// TIA Portal V19 export
DATA_BLOCK "DB_NSP"   // DB96
{ S7_Optimized_Access := 'FALSE' }
// stored: AutoNumber false
   VAR RETAIN
      Anz_Per_Cyc : Int := 10;   // * Anzahl Positionen pro Zyklus (kleiner eine Sekunde müssen alle durch sein)
      Offset : Int := 20;   // Beginn Datenblock
      leng : Int := 20;   // Länge einer Struktue
      akt_NSP : Int := 55;   // aktueller Eintrag
      Test_on : Bool := TRUE;   // Testfunktion aktiv (nicht gewählte NSP/SPR aus)
      Test_akt : Bool := FALSE;   // Test Einzelpos (TestNr) aktiv
      Test_start : Bool := FALSE;   // Test angemeldet erster Umlauf alles aus
      Sekunde : Bool := FALSE;   // Sekunde M2.5 war ein
      Takt : Bool := FALSE;   // Takt (Sekunde) Zeiten zählen
      AMS_Reset : Bool := FALSE;   // Reset gefordert
      AMS_new : Bool := FALSE;   // Meldung neu schicken
      SammelWarn : Bool := FALSE;   // SammelWarnung min/max über alle Pos.
      Sammelstoer : Bool := FALSE;   // Sammelstörung Timeout über alle Pos.
      noMD_opt_max : Bool := FALSE;   // Überlauf nicht optisch melden
      noMD_opt_min : Bool := FALSE;   // Niveau min nicht optisch melden
      noMD_opt_Zeit : Bool := FALSE;   // Zeitüberschreit. nicht optisch melden
      noMD_aku_max : Bool := FALSE;   // Überlauf nicht akustisch melden
      noMD_aku_min : Bool := FALSE;   // Niveau min nicht akustisch melden
      noMD_aku_Zeit : Bool := FALSE;   // Zeitüberschreit. nicht akustisch melden
      Reset : Bool := FALSE;   // Reset Timeout NS
      TestNr : Int := 0;   // Nachspeisung für Test (alle anderen werden nicht bearbeitet)
      temp_Warn : Bool := FALSE;
      temp_STM : Bool := FALSE;
      resX122 : Bool := FALSE;
      resX123 : Bool := FALSE;
      resX124 : Bool := FALSE;
      resX125 : Bool := FALSE;
      resX126 : Bool := FALSE;
      resX127 : Bool := FALSE;
      resB1 : Byte := 16#00;
      resW1 : Int := 0;
      resD1 : DInt := 0;
      NSP : Array[1..30] of Struct
         NSP : Bool;   // Niveauregelung
         NST_in : Bool;   // Takt nach WT im Bad eingesetzt
         NST_out : Bool;   // Takt nach WT aus Bad ausgehoben
         SPR_in : Bool;   // Spritzen bei FW senkt
         SPR_out : Bool;   // Spritzen bei FW hebt
         SPR_expo : Bool;   // Spritzen während Expozeit
         SPR_Zeit : Bool;   // Spritzen feste Zeit nach Ausheben oder Einsetzen
         resTyp1 : Bool;   // ReserveTyp
         resTyp2 : Bool;   // ReserveTyp
         resTyp3 : Bool;   // ReserveTyp
         resTyp4 : Bool;   // ReserveTyp
         resTyp5 : Bool;   // ReserveTyp
         resTyp6 : Bool;   // ReserveTyp
         resTyp7 : Bool;   // ReserveTyp
         resTyp8 : Bool;   // ReserveTyp
         resTyp9 : Bool;   // ReserveTyp
         Freigabe : Bool;   // Freigabe Nachspeisung
         extern_Start : Bool;   // externe Aktivierung Taktung (zum Beispiel bei mehreren Pos)
         Niveau_ok : Bool;   // Niveau is ok Nachspeisung über Niveauregelung aus
         Nachspeisen : Bool;   // Nachspeisung aktiv --> Ventil auf / Pumpe an
         Spritzen : Bool;   // Spritzregister ein
         AL_Ueberlauf : Bool;   // Behälter Überlauf
         AL_Niv_min : Bool;   // Niveau zu niedrig --> Behälter leer
         AL_Zeit : Bool;   // Nachspeise-Zeitüberschreitung
         Restzeit_NSP : Int;   // Restzeit Nachspeisung
         TestNSP : Int;   // Testzeit Nachspeisung
         Restzeit_SPR : Int;   // Restzeit Spritzen
         VerzT : Int;   // Verzögerung Alarm Überlauf/Min-Niveau
         RestVerz : Int;   // Restzeit bis Alarm
         VerzNS_AL : Int;   // Verzögerung Alarm Nachspeisezeit zu gross
         RestNS_AL : Int;   // Restzeit bis Alarm
         AM_AL_min : Bool;   // Altmerker Alarm min
         AM_AL_Uel : Bool;   // Altmerker Alarm voll
         AM_AL_Zeit : Bool;   // Altmerker Alarm Nachspeise-Zeitüberschreitung
         AM_Bad_belegt : Bool;   // Altmerker Bad belegt
         AM_Reset : Bool;   // Altmerker RESET Nachspeise-Zeitüberschreitung
         res2 : Bool;
         res3 : Bool;
         res4 : Bool;
         SprFree : Bool;   // Spritzregister nicht bedienen (keine Ausgabe weder on noch off) Bedienung ext.
         NSPFree : Bool;   // Nachspeisung nicht bedienen (keine Ausgabe weder on noch off) Bedienung extern
         Warte_NSPT : Bool;   // getaktete Nachspeisung nicht abarbeiten
         res8 : Bool;
         res9 : Bool;
         res10 : Bool;
         res11 : Bool;
         res12 : Bool;
      END_STRUCT;
   END_VAR
BEGIN
   NSP[1..30].NSP := FALSE;
   NSP[1..30].NST_in := FALSE;
   NSP[1..30].NST_out := FALSE;
   NSP[1..30].SPR_in := FALSE;
   NSP[1..25].SPR_out := FALSE;
   NSP[26].SPR_out := TRUE;
   NSP[27..29].SPR_out := FALSE;
   NSP[30].SPR_out := TRUE;
   NSP[1..30].SPR_expo := FALSE;
   NSP[1..30].SPR_Zeit := FALSE;
   NSP[1..30].resTyp1 := FALSE;
   NSP[1..30].resTyp2 := FALSE;
   NSP[1..30].resTyp3 := FALSE;
   NSP[1..30].resTyp4 := FALSE;
   NSP[1..30].resTyp5 := FALSE;
   NSP[1..30].resTyp6 := FALSE;
   NSP[1..30].resTyp7 := FALSE;
   NSP[1..30].resTyp8 := FALSE;
   NSP[1..30].resTyp9 := FALSE;
   NSP[1..30].Freigabe := FALSE;
   NSP[1..30].extern_Start := FALSE;
   NSP[1..30].Niveau_ok := FALSE;
   NSP[1..30].Nachspeisen := FALSE;
   NSP[1..30].Spritzen := FALSE;
   NSP[1..30].AL_Ueberlauf := FALSE;
   NSP[1..30].AL_Niv_min := FALSE;
   NSP[1..30].AL_Zeit := FALSE;
   NSP[1..30].Restzeit_NSP := 0;
   NSP[1..30].TestNSP := 0;
   NSP[1..30].Restzeit_SPR := 0;
   NSP[1..30].VerzT := 0;
   NSP[1..30].RestVerz := 0;
   NSP[1..30].VerzNS_AL := 0;
   NSP[1..30].RestNS_AL := 0;
   NSP[1..30].AM_AL_min := FALSE;
   NSP[1..30].AM_AL_Uel := FALSE;
   NSP[1..30].AM_AL_Zeit := FALSE;
   NSP[1..30].AM_Bad_belegt := FALSE;
   NSP[1..30].AM_Reset := FALSE;
   NSP[1..30].res2 := FALSE;
   NSP[1..30].res3 := FALSE;
   NSP[1..30].res4 := FALSE;
   NSP[1..30].SprFree := FALSE;
   NSP[1..30].NSPFree := FALSE;
   NSP[1..30].Warte_NSPT := FALSE;
   NSP[1..30].res8 := FALSE;
   NSP[1..30].res9 := FALSE;
   NSP[1..30].res10 := FALSE;
   NSP[1..30].res11 := FALSE;
   NSP[1..30].res12 := FALSE;
END_DATA_BLOCK
